FUNCTION_BLOCK FB_AnlgSIM
VAR_INPUT
	Mn:REAL;
	Mx:REAL;
END_VAR

VAR_OUTPUT
END_VAR
VAR_IN_OUT
	Sen:REAL;
END_VAR
VAR
	timInc : TON;
	timRst : TON;
	timInc2 : TON;
	incVal:INT:=100;
END_VAR


IF timInc.Q THEN
	IF Sen >= Mx-incVal THEN
		timRst(IN:=TRUE,PT:=T#1S);
		IF timRst.Q THEN
			timRst(IN:=FALSE);
			Sen := Mn; 
		END_IF
	ELSE
		IF Sen=Mn THEN
			timInc2(IN:=TRUE,PT:=T#1S);	
			IF timInc2.Q THEN
				timInc2(IN:=FALSE);
					Sen := Sen+incVal;
			END_IF
		ELSE
			IF Sen >=Mx-incVal THEN
			    Sen := Mx-incVal;
			ELSE
				Sen := Sen+incVal; 
			END_IF 
		END_IF
	END_IF
	timInc(IN:=FALSE);
ELSE
	timInc(IN:=TRUE,PT:=T#40MS);
END_IF

END_FUNCTION_BLOCK

(* stored: Version 1.1.0.1, ProductVersion 3.1.4022.18
   POU FB_AnlgSIM: Id {ad10ddd2-3c62-4914-a9a7-47aaa096944f}, SpecialFunc None *)
